// TwinCAT 3 PLC project HydroValve
// ProgramVersion: 3.1.4024.0
// libraries:
//   Tc2_Standard, * (Beckhoff Automation GmbH)
//   Tc2_System, * (Beckhoff Automation GmbH)
//   Tc3_Module, * (Beckhoff Automation GmbH)
// project tree:
//   DUTs/ configaracionParammetrs.TcDUT, errorsSt.TcDUT, Staus.TcDUT, StrRampTime.TcDUT
//   GVLs/ generalVariable.TcGVL (not stored)
//   / PlcTask.TcTTO
//   POUs/ acc_dec.TcPOU, acc_dec_Valve.TcPOU, blockMessage.TcPOU, MAIN.TcPOU, Monitoring_Error.TcPOU, Solenoid.TcPOU, HydraulicValve.TcPOU
//   POUs/convert/ convertToAm.TcPOU, convertToHodnota.TcPOU
// real-time tasks:
//   TASK PlcTask: cycle T#10ms, priority 20, ADS port 350

CONFIGURATION HydroValve
    RESOURCE PLC ON TwinCAT3
        TASK PlcTask(INTERVAL := T#10ms, PRIORITY := 20);
        PROGRAM MAIN WITH PlcTask : MAIN;
    END_RESOURCE
END_CONFIGURATION

// ---- DUTs/configaracionParammetrs.TcDUT
TYPE configaracionParammetrs :
STRUCT
	CurPosDirMin : REAL := 100; // Minimální proud na solenoid v daném směru [mA]
	CurPosDirMax : REAL := 500; // Maximální proud na solenoid v daném směru [mA]
	CurNegDirMin : REAL := 100; // Minimální proud na solenoid v daném směru [mA]
	CurNegDirMax : REAL := 500; // Maximální proud na solenoid v daném směru [mA]
	RampPosDirUp : INT := 100; // Doba změny z min. na max. otevření v daném směru [ms]
	RampPosDirDown :INT := 100; // Doba změny z max. na min. otevření v daném směru [ms]
	RampNegDirUp : INT := 100; // Doba změny z min. na max. otevření v daném směru [ms]
	RampNegDirDown : INT := 100; // Doba změny z max. na min. otevření v daném směru [ms]
	Deadtime : TIME := T#5MS; // Kompenzace setrvačnosti při reverzaci [ms]
END_STRUCT
END_TYPE

// ---- DUTs/errorsSt.TcDUT
TYPE errorsSt :
STRUCT
	errorName	:	STRING;
	showError	:	BOOL;
END_STRUCT
END_TYPE

// ---- DUTs/Staus.TcDUT
TYPE Staus :
STRUCT
	Standstill : BOOL;	// Oba výstupy jsou na minimu
	Accel : BOOL;	// Jeden z výstupů zrychluje
	Decel : BOOL;	// Jeden z výstupů zpomaluje
	OutPosDirProc : REAL;// Výstup v daném směru [%]
	OutNegDirProc : REAL;// Výstup v daném směru [%]
	bBussy : BOOL;// TRUE je-li FB aktivní (změna na výstupu)
	bDone : BOOL;	// TRUE je-li výstupní hodnota je rovna žádané
	bError : ARRAY[1..50] OF errorsSt; // Chyba
	nErrorId : ARRAY[1..50] OF INT;// Kód chyby
END_STRUCT
END_TYPE

// ---- DUTs/StrRampTime.TcDUT
TYPE StrRampTime :
STRUCT
	rampTimeNegMaxMin	:	TIME;
	rampTimeNegMinMax	:	TIME;
	rampTimePosMaxMin	:	TIME;
	rampTimePosMinMax	:	TIME;
END_STRUCT
END_TYPE

// ---- POUs/MAIN.TcPOU
PROGRAM MAIN
VAR
	hydValve : HydraulicValve();
	monError	:	Monitoring_Error();
	enaNegDirB : BOOL := FALSE;
	enaPosDirB : BOOL := FALSE;
	commandSet : REAL := 0;
	currentError	:	BOOL := FALSE;
	//konfiguraParametry : REFERENCE TO configaracionParammetrs  REF=generalVariable.conParammetr;
	OutPosDir : REAL := 0 ;	// Výstup v daném směru [mA]
	OutNegDir : REAL := 0 ;	// Výstup v daném směru [mA]
END_VAR

IF NOT(generalVariable.staus.bBussy) THEN
	monError(negDirB := enaNegDirB, posDirB := enaPosDirB, command := commandSet);
	IF NOT(monError.currentError) THEN
		hydValve(bvNegDir := enaNegDirB, bvPosDir := enaPosDirB, command := commandSet); 
	END_IF
END_IF
OutPosDir := convertToAm(generalVariable.staus.OutPosDirProc * 10, TRUE);
OutNegDir := convertToAm(generalVariable.staus.OutNegDirProc * 10, FALSE);

END_PROGRAM

// ---- POUs/HydraulicValve.TcPOU
FUNCTION_BLOCK HydraulicValve
VAR_INPUT
	bvPosDir	: BOOL;
	bvNegDir	: BOOL;
	command		: REAL;
END_VAR
VAR
	rampTimeACC	: REAL;
	rampTimeDEC	: REAL;
	curentSolenoid	:	SINT;	// neg -1, pos 1, nobady 0
	posDir	:	Solenoid();
	negDir	:	Solenoid(); 
END_VAR
VAR_OUTPUT
	OutPosDir : REAL := 0 ;	// Výstup v daném směru [mA]
	OutNegDir : REAL := 0 ;	// Výstup v daném směru [mA]
END_VAR

curentSolenoid := howIsActive();

CASE curentSolenoid OF
	1	:	posDir( desiredPosition := command, bPosDir := bvPosDir);
	-1	:	negDir(desiredPosition := command, bPosDir := bvPosDir);
	0	:	daethTime(dTime := generalVariable.conParammetr.Deadtime);
			IF bvPosDir THEN
				posDir( desiredPosition := command, bPosDir := bvPosDir);
				ELSIF bvNegDir THEN
					negDir(desiredPosition := command, bPosDir := bvPosDir);
					END_IF;
END_CASE
//generalVariable.staus.OutPosDirProc := posDir.OutDir;
OutPosDir := posDir.OutDir;
OutNegDir := negDir.OutDir;

METHOD PRIVATE daethTime 
VAR_INPUT
	dTime	:	TIME;
END_VAR
VAR
	
	wait_death_time	:	TON;
END_VAR
dTime := generalVariable.conParammetr.Deadtime;
acc_dec(FALSE, FALSE);
generalVariable.staus.Standstill := TRUE;
wait_death_time(IN:=TRUE , PT:=dTime , Q=> , ET=> );
END_METHOD

METHOD howIsActive : SINT
VAR_INPUT
END_VAR
IF (posDir.OutDir > 0) THEN
	howIsActive := 1;
	generalVariable.staus.OutPosDirProc := posDir.OutDir/10;
	generalVariable.staus.OutNegDirProc := 0;
	ELSIF (negDir.OutDir < 0) THEN
		howIsActive := -1;
		generalVariable.staus.OutPosDirProc := 0;
		generalVariable.staus.OutNegDirProc := negDir.OutDir/10;
		ELSE
			howIsActive := 0;
			END_IF;
END_METHOD

METHOD PRIVATE RampTimeNeg : REAL
IF bvPosDir THEN
	rampTimeACC:= generalVariable.conParammetr.CurNegDirMax/generalVariable.conParammetr.RampNegDirUp;
	ELSE
		rampTimeDEC := generalVariable.conParammetr.CurNegDirMin/generalVariable.conParammetr.RampNegDirDown;
		END_IF;
END_METHOD

METHOD PRIVATE RampTimePos : REAL
IF bvPosDir THEN
	rampTimeACC := (generalVariable.conParammetr.CurPosDirMax/generalVariable.conParammetr.RampPosDirUp);
	ELSE
		rampTimeDEC := (generalVariable.conParammetr.CurPosDirMin/generalVariable.conParammetr.RampPosDirDown);
		END_IF;
END_METHOD

END_FUNCTION_BLOCK

// ---- POUs/Solenoid.TcPOU
FUNCTION_BLOCK Solenoid
VAR_INPUT
	desiredPosition	:	REAL;
	bPosDir			:	BOOL;
END_VAR
VAR
	curPosition		:	REAL;
	rampTime		:	StrRampTime;
	loc_rampTime	:	TIME;
	delta			:	REAL;
END_VAR
VAR_OUTPUT
	OutDir : REAL;	// Výstup v daném směru 
END_VAR

RampTimeMethod(desiredPosition, curPosition);
curPosition := desiredPosition;
IF (curPosition * desiredPosition >= 0) THEN
			// na istom solenoidu
			IF (ABS(desiredPosition) > ABS(curPosition)) THEN
			    // ACC
				IF (curPosition > 0) THEN
					loc_rampTime := rampTime.rampTimePosMinMax;
					ELSE
						loc_rampTime := rampTime.rampTimeNegMinMax;
						END_IF;
				// DEC
				ELSIF (curPosition > 0) THEN					
					loc_rampTime := rampTime.rampTimePosMaxMin;
					ELSE
						loc_rampTime := rampTime.rampTimeNegMaxMin;
						END_IF;
				curPosition := acc_dec_Valve(requiredValue := desiredPosition, currentValue := curPosition, rampTime := loc_rampTime);
			ELSE  
				//postoji prelaz
				blockMessage('Postoji prelaz');
				IF (curPosition >= 0) THEN
					curPosition := acc_dec_Valve(requiredValue := 0, currentValue := curPosition, rampTime := RampTime.rampTimePosMinMax);
					ELSE
						curPosition := acc_dec_Valve(requiredValue := 0, currentValue := curPosition, rampTime := RampTime.rampTimeNegMaxMin);
						END_IF;
					
			END_IF;

OutDir := curPosition;

METHOD PRIVATE RampTimeMethod
VAR
	razlika	:	REAL;
END_VAR
VAR_INPUT
	desiredPosition	:	REAL;
	curPosition		:	REAL;
END_VAR

razlika := convertToAm((desiredPosition - curPosition), bPosDir);
rampTime.rampTimeNegMaxMin := REAL_TO_TIME(razlika / (generalVariable.conParammetr.CurNegDirMax/generalVariable.conParammetr.RampNegDirUp));
rampTime.rampTimeNegMinMax := REAL_TO_TIME(razlika / (generalVariable.conParammetr.CurNegDirMin/generalVariable.conParammetr.RampNegDirDown));
rampTime.rampTimePosMaxMin := REAL_TO_TIME(razlika / (generalVariable.conParammetr.CurPosDirMax/generalVariable.conParammetr.RampPosDirUp));
rampTime.rampTimePosMinMax := REAL_TO_TIME(razlika / (generalVariable.conParammetr.CurPosDirMin/generalVariable.conParammetr.RampPosDirDown));
END_METHOD

END_FUNCTION_BLOCK

// ---- POUs/acc_dec_Valve.TcPOU
FUNCTION acc_dec_Valve : REAL
VAR_INPUT
		requiredValue	:	REAL;
		currentValue	:	REAL;
		rampTime		:	TIME;
END_VAR
VAR
	delta	:	REAL;
END_VAR


generalVariable.staus.bBussy := TRUE;
generalVariable.staus.bDone := FALSE;
delta := ABS(requiredValue) - ABS(currentValue);
IF (delta > 0) THEN
	acc_dec(TRUE, FALSE);
	currentValue := currentValue + (requiredValue -currentValue) * _TaskInfo[GETCURTASKINDEXEX()].CycleTime/TIME_TO_REAL(rampTime);
	ELSE
		acc_dec(FALSE, TRUE);
		acc_dec_Valve := currentValue + (requiredValue -currentValue) * _TaskInfo[GETCURTASKINDEXEX()].CycleTime/TIME_TO_REAL(rampTime);
	END_IF;
	
IF (requiredValue >= currentValue) THEN
	requiredValue := currentValue;
	acc_dec(FALSE, FALSE);	
	generalVariable.staus.bBussy := FALSE;
	generalVariable.staus.bDone := TRUE;
END_IF

END_FUNCTION

// ---- POUs/acc_dec.TcPOU
FUNCTION acc_dec : bool
VAR_INPUT
	a	:	BOOL;
	d	:	BOOL;
END_VAR
VAR
END_VAR

generalVariable.staus.Accel := a;
generalVariable.staus.Decel := d;

END_FUNCTION

// ---- POUs/blockMessage.TcPOU
FUNCTION blockMessage 
VAR_INPUT
	error : STRING;
	
END_VAR
VAR
	strSFCErrorStep : STRING; (* Declaration*)
END_VAR

//	writing messages, help for me
ADSLOGSTR(msgCtrlMask := ADSLOG_MSGTYPE_ERROR OR ADSLOG_MSGTYPE_LOG,
	msgFmtStr := error,
	strArg := strSFCErrorStep);

END_FUNCTION

// ---- POUs/convert/convertToAm.TcPOU
FUNCTION convertToAm : REAL
VAR_INPUT
	pCommand	:	REAL;
	enaPosDir	:	BOOL;
END_VAR
VAR
END_VAR


IF  enaPosDir THEN
	convertToAm:= (ABS(pCommand) * (generalVariable.conParammetr.CurPosDirMax - generalVariable.conParammetr.CurPosDirMin)/1000) + generalVariable.conParammetr.CurPosDirMin;
	ELSE
		convertToAm:= (ABS(pCommand) * (generalVariable.conParammetr.CurNegDirMax - generalVariable.conParammetr.CurNegDirMin)/1000) + generalVariable.conParammetr.CurNegDirMin;
		END_IF;

END_FUNCTION

// ---- POUs/Monitoring_Error.TcPOU
FUNCTION_BLOCK Monitoring_Error
VAR_INPUT
	negDirB	:	BOOL;
	posDirB	:	BOOL;
	command	:	REAL;
END_VAR
VAR_OUTPUT
	currentError	:	BOOL;
END_VAR

// list errors on inout 
enableSolenoidControl(enaNegDir := negDirB, enaPosDir := posDirB, error := currentError);
commandCheck(comm := command, error := currentError);

METHOD PRIVATE commandCheck
VAR_INPUT
	comm : REAL;
END_VAR
VAR_IN_OUT
	error: BOOL;
END_VAR
// control command and enaeble direction
IF ((comm <= 1000) AND (comm >0)) THEN
		IF posDirB THEN
			error := FALSE;
			generalVariable.staus.bError[2].showError := FALSE;
			ELSE
				error := TRUE;
				showError(2,'příkaz a směr se neshodují');
				END_IF;
	ELSIF ((comm >= -1000) AND (comm < 0)) THEN
			IF negDirB THEN
				error := FALSE;
				generalVariable.staus.bError[2].showError := FALSE;
			ELSE
				error := TRUE;
				showError(2,'příkaz a směr se neshodují');
				END_IF;
			ELSIF comm = 0 THEN
				generalVariable.staus.Standstill := TRUE;
				IF NOT(negDirB AND posDirB) THEN
					error := FALSE;
					generalVariable.staus.bError[3].showError := FALSE;
				ELSE
					error := TRUE;
					showError(3,'zahrnoval některé směry');       
				END_IF;
			END_IF;
END_METHOD

METHOD PRIVATE enableSolenoidControl
VAR_INPUT
	enaPosDir : BOOL;
	enaNegDir : BOOL;	
END_VAR
VAR_IN_OUT
	error: BOOL;
END_VAR
VAR
	strr	:	STRING;
END_VAR
//	control enaeble direction
IF (enaNegDir AND enaPosDir) THEN
	// error 
	currentError := TRUE;
	showError(1,'muze být aktivní pouze jedna cívka (PosDir nebo NegDir)');
	//errCode(1);
	ELSE
		currentError := FALSE ;
		generalVariable.staus.bError[1].showError := FALSE;
		END_IF
END_METHOD

METHOD PRIVATE showError
VAR_INPUT
	id	:	INT;
	str	:	STRING;
END_VAR
//	show errora
generalVariable.staus.bError[50].showError := FALSE;
IF NOT(generalVariable.staus.bError[id].showError) THEN
	generalVariable.staus.nErrorId[id] := id;
	generalVariable.staus.bError[id].errorName := str;
	generalVariable.staus.bError[id].showError := TRUE;
	blockMessage(str);
	END_IF;
END_METHOD

END_FUNCTION_BLOCK

// ---- POUs/convert/convertToHodnota.TcPOU
FUNCTION convertToHodnota : REAL

VAR_INPUT
	pCommand	:	REAL;
	enaPosDir	:	BOOL;
END_VAR

//	mA  conversion  in  0 to 1000
IF  enaPosDir THEN
	convertToHodnota := (pCommand * (generalVariable.conParammetr.CurPosDirMax - generalVariable.conParammetr.CurPosDirMin)/1000) + generalVariable.conParammetr.CurPosDirMin;
	ELSE
		convertToHodnota := (pCommand * (generalVariable.conParammetr.CurNegDirMax - generalVariable.conParammetr.CurNegDirMin)/1000) + generalVariable.conParammetr.CurNegDirMin;
		END_IF;

END_FUNCTION
